// TIA Portal V16 export
// export: Created 2021-10-20T14:42:06.6500915Z, ExportSetting WithDefaults, DisplayName Totally Integrated Automation Portal, DisplayVersion V16, DisplayName TIA Portal Version Control Interface, DisplayVersion V16, DisplayName TIA Portal Openness, DisplayVersion V16, DisplayName TIA Portal Teamcenter Gateway, DisplayVersion V16, DisplayName SINAMICS Startdrive Advanced, DisplayVersion V16, DisplayName SINAMICS Startdrive G130, G150, S120, S150, SINAMICS MV, S210, DisplayVersion V16, DisplayName SINAMICS Startdrive G110M, G120, G120C, G120D, G120P, DisplayVersion V16, DisplayName STEP 7 Professional, DisplayVersion V16, DisplayName STEP 7 Safety, DisplayVersion V16, DisplayName WinCC Advanced, DisplayVersion V16
FUNCTION_BLOCK "Faults"   // FB5, LAD
TITLE = Faults
{ S7_Optimized_Access := 'TRUE' }
VERSION : 0.1
// stored: AutoNumber true, IsIECCheckEnabled false, IsRetainMemResEnabled false, MemoryReserve 100, SetENOAutomatically false, UDAEnableTagReadback false
BEGIN

REGION Network 1: Rm4 Air Flow Fault
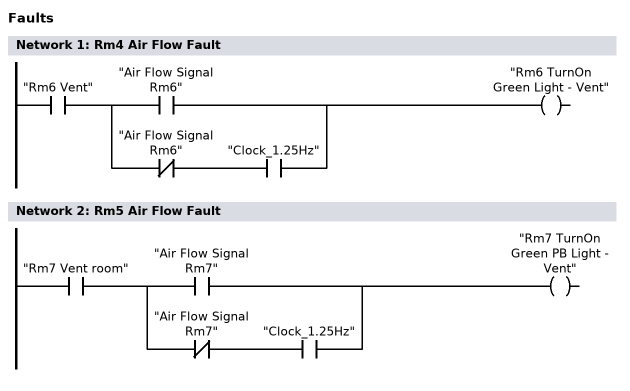
   RUNG wire#powerrail
      Contact( "Rm6 Vent" )
      wire#w1
      Contact( "Air Flow Signal Rm6" )
      wire#w2
      Coil( "Rm6 TurnOn Green Light - Vent" )
   END_RUNG
   RUNG wire#w1
      I_Contact( "Air Flow Signal Rm6" )
      Contact( "Clock_1.25Hz" )
   END_RUNG wire#w2
   // the same network as SCL:
   "Rm6 TurnOn Green Light - Vent" := "Rm6 Vent" AND ("Air Flow Signal Rm6" OR (NOT "Air Flow Signal Rm6" AND "Clock_1.25Hz"));
END_REGION

REGION Network 2: Rm5 Air Flow Fault
   RUNG wire#powerrail
      Contact( "Rm7 Vent room" )
      wire#w1
      Contact( "Air Flow Signal Rm7" )
      wire#w2
      Coil( "Rm7 TurnOn Green PB Light - Vent" )
   END_RUNG
   RUNG wire#w1
      I_Contact( "Air Flow Signal Rm7" )
      Contact( "Clock_1.25Hz" )
   END_RUNG wire#w2
   // the same network as SCL:
   "Rm7 TurnOn Green PB Light - Vent" := "Rm7 Vent room" AND ("Air Flow Signal Rm7" OR (NOT "Air Flow Signal Rm7" AND "Clock_1.25Hz"));
END_REGION
END_FUNCTION_BLOCK
